DATA_BLOCK "Auto_DB"
{ S7_Optimized_Access := 'TRUE' }
VERSION : 0.1
NON_RETAIN
"Auto"

BEGIN

END_DATA_BLOCK

